FUNCTION_BLOCK MIN_REAL (* IEC 61131-3 REAL Minimum *)
  (* Standard: 61131-3 *)
  (* Version 0.0, 2004-12-15, JHC, Rockwell Automation, Converted from SRC format. *)
  (* Compiler header: package fb.rt.plc.select; *)
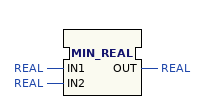
  VAR_INPUT
    IN1 : REAL;
    IN2 : REAL;
  END_VAR
  VAR_OUTPUT
    OUT : REAL; (* MIN(IN1,IN2) *)
  END_VAR
END_FUNCTION_BLOCK
